// TIA Portal V20 export
TYPE "typeCmHmiInterfaceSoftCamjrOutPnPRightAxisZ"
// stored: Access Published, Namespace Unit1.Em2
   STRUCT
      pos00_wait : "LER_typeSoftCamPosition";
      pos01_load : "LER_typeSoftCamPosition";
      pos02_unload : "LER_typeSoftCamPosition";
      pos03_posistion { ExternalWritable := 'False'} : "LER_typeSoftCamPosition";
      pos04_posistion { ExternalWritable := 'False'} : "LER_typeSoftCamPosition";
      pos05_posistion { ExternalWritable := 'False'} : "LER_typeSoftCamPosition";
      pos06_posistion { ExternalWritable := 'False'} : "LER_typeSoftCamPosition";
      pos07_posistion { ExternalWritable := 'False'} : "LER_typeSoftCamPosition";
      pos08_posistion { ExternalWritable := 'False'} : "LER_typeSoftCamPosition";
      pos09_noInterferenceZone : "LER_typeSoftCamPosition";
      pos10_posistion { ExternalWritable := 'False'} : "LER_typeSoftCamPosition";
      pos11_posistion { ExternalWritable := 'False'} : "LER_typeSoftCamPosition";
      pos12_posistion { ExternalWritable := 'False'} : "LER_typeSoftCamPosition";
      pos13_posistion { ExternalWritable := 'False'} : "LER_typeSoftCamPosition";
      pos14_posistion { ExternalWritable := 'False'} : "LER_typeSoftCamPosition";
      pos15_posistion { ExternalWritable := 'False'} : "LER_typeSoftCamPosition";
   END_STRUCT;
END_TYPE
